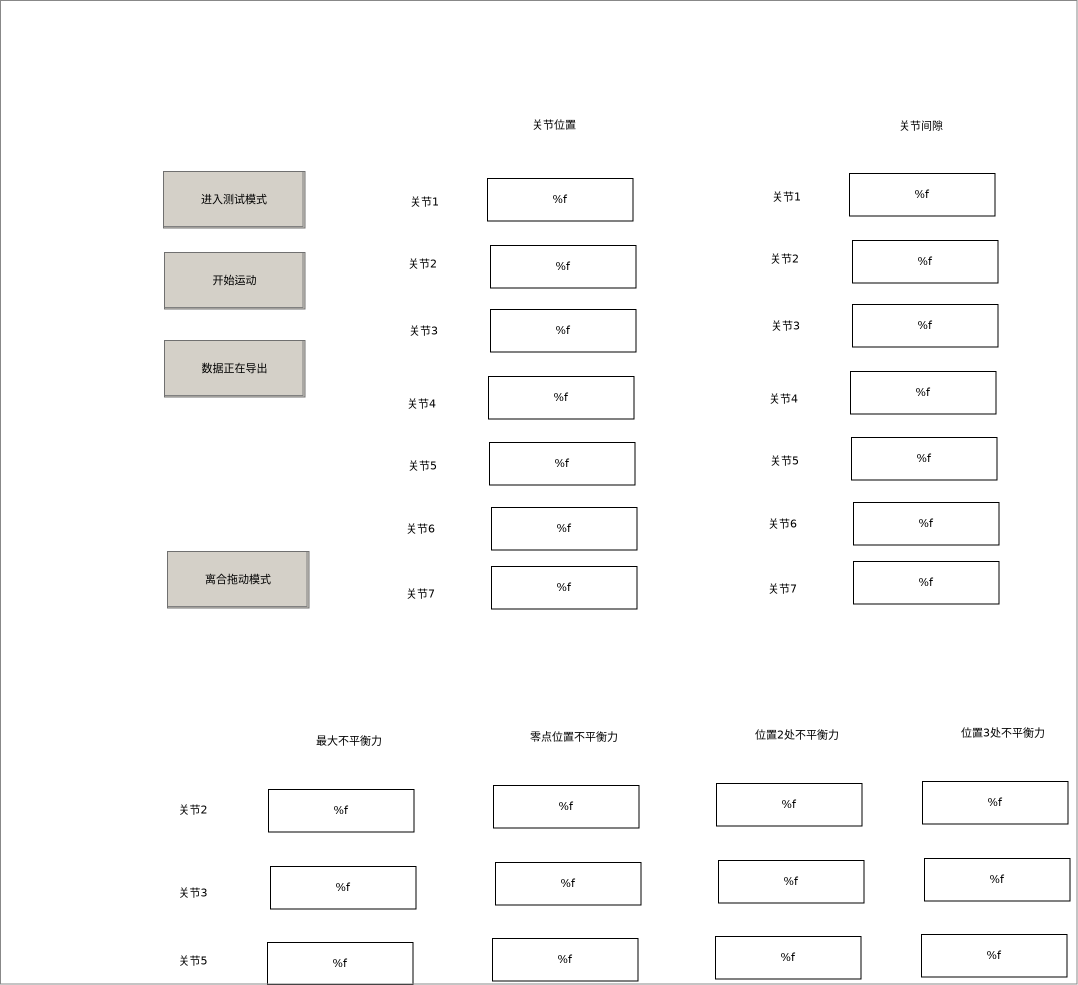
VISUALIZATION armTest  // 1078x985
    Button (163,171 142x57), "进入测试模式", colour toggle: GVL_armTest.g_testMode[1]
        toggle GVL_armTest.g_testMode[1]
    Button (164,252 141x57), "开始运动", colour toggle: GVL_armTest.g_startMotion[1]
        toggle GVL_armTest.g_startMotion[1]
    Rectangle (487,178 146x43), "%f", text variable: GVL_armTest.g_armDHJntPos[1][1]
    Label (373,184 103x36), "关节1"
    Label (371,246 103x36), "关节2"
    Label (372,313 103x36), "关节3"
    Label (370,386 103x36), "关节4"
    Label (371,448 103x36), "关节5"
    Label (369,511 103x36), "关节6"
    Label (369,576 103x36), "关节7"
    Rectangle (490,245 146x43), "%f", text variable: GVL_armTest.g_armDHJntPos[1][2]
    Rectangle (490,309 146x43), "%f", text variable: GVL_armTest.g_armDHJntPos[1][3]
    Rectangle (488,376 146x43), "%f", text variable: GVL_armTest.g_armDHJntPos[1][4]
    Rectangle (489,442 146x43), "%f", text variable: GVL_armTest.g_armDHJntPos[1][5]
    Rectangle (491,507 146x43), "%f", text variable: GVL_armTest.g_armDHJntPos[1][6]
    Rectangle (491,566 146x43), "%f", text variable: GVL_armTest.g_armDHJntPos[1][7]
    Button (167,551 142x57), "离合拖动模式", colour toggle: GVL_armTest.g_clutchMode[1]
        toggle GVL_armTest.g_clutchMode[1]
    Rectangle (849,173 146x43), "%f", text variable: GVL_armTest.g_jntGap[1][1]
    Label (735,179 103x36), "关节1"
    Label (733,241 103x36), "关节2"
    Label (734,308 103x36), "关节3"
    Label (732,381 103x36), "关节4"
    Label (733,443 103x36), "关节5"
    Label (731,506 103x36), "关节6"
    Label (731,571 103x36), "关节7"
    Rectangle (852,240 146x43), "%f", text variable: GVL_armTest.g_jntGap[1][2]
    Rectangle (852,304 146x43), "%f", text variable: GVL_armTest.g_jntGap[1][3]
    Rectangle (850,371 146x43), "%f", text variable: GVL_armTest.g_jntGap[1][4]
    Rectangle (851,437 146x43), "%f", text variable: GVL_armTest.g_jntGap[1][5]
    Rectangle (853,502 146x43), "%f", text variable: GVL_armTest.g_jntGap[1][6]
    Rectangle (853,561 146x43), "%f", text variable: GVL_armTest.g_jntGap[1][7]
    Label (479,110 150x30), "关节位置"
    Label (846,111 150x30), "关节间隙"
    Label (118,795 150x30), "关节2"
    Label (118,878 150x30), "关节3"
    Label (118,946 150x30), "关节5"
    Rectangle (268,789 146x43), "%f", text variable: GVL_armTest.g_unbalancedMax[1][2]
    Label (274,726 150x30), "最大不平衡力"
    Rectangle (270,866 146x43), "%f", text variable: GVL_armTest.g_unbalancedMax[1][3]
    Rectangle (267,942 146x43), "%f", text variable: GVL_armTest.g_unbalancedMax[1][5]
    Rectangle (493,785 146x43), "%f", text variable: GVL_armTest.g_jntTestPntUnbalancedTrq[1,2,1]
    Label (499,722 150x30), "零点位置不平衡力"
    Rectangle (495,862 146x43), "%f", text variable: GVL_armTest.g_jntTestPntUnbalancedTrq[1,3,1]
    Rectangle (492,938 146x43), "%f", text variable: GVL_armTest.g_jntTestPntUnbalancedTrq[1,5,1]
    Rectangle (716,783 146x43), "%f", text variable: GVL_armTest.g_jntTestPntUnbalancedTrq[1,2,2]
    Label (722,720 150x30), "位置2处不平衡力"
    Rectangle (718,860 146x43), "%f", text variable: GVL_armTest.g_jntTestPntUnbalancedTrq[1,3,2]
    Rectangle (715,936 146x43), "%f", text variable: GVL_armTest.g_jntTestPntUnbalancedTrq[1,5,2]
    Rectangle (922,781 146x43), "%f", text variable: GVL_armTest.g_jntTestPntUnbalancedTrq[1,2,3]
    Label (928,718 150x30), "位置3处不平衡力"
    Rectangle (924,858 146x43), "%f", text variable: GVL_armTest.g_jntTestPntUnbalancedTrq[1,3,3]
    Rectangle (921,934 146x43), "%f", text variable: GVL_armTest.g_jntTestPntUnbalancedTrq[1,5,3]
    Button (164,340 141x57), "数据正在导出", colour toggle: GVL_armTest.g_duringWriteData[1]
END_VISUALIZATION

(* stored: Version 1.1.0.1, ProductVersion 3.1.4024.11
   Visu armTest: Id {831c13d7-b138-4dce-bd94-5dfa665395e3} *)
